FUNCTION_BLOCK FB_Scale
VAR_INPUT
    nRaw : DINT;            // counts from the load cell terminal
END_VAR
VAR
    fWeight     : LREAL;    // g
    fLastWeight : LREAL;
END_VAR

fLastWeight := fWeight;
fWeight := DINT_TO_LREAL(nRaw) * 0.01;

PROPERTY IsSettled : BOOL
GET
IsSettled := (fWeight = fLastWeight);
END_GET
END_PROPERTY

END_FUNCTION_BLOCK

(* stored: Version 1.1.0.1, ProductVersion 3.1.4024.0
   POU FB_Scale: Id {11ccd30e-da70-4526-852d-ad83462883d6}, SpecialFunc None
   Property IsSettled: Id {ca61f444-9247-4388-8494-115e6f29389a}
   Get Get: Id {ae162878-a7d8-4aa0-b391-f563ff084c0d} *)
